INTERFACE I_Pneumatic EXTENDS I_Device

METHOD cancel : BOOL
VAR_INPUT
END_VAR
END_METHOD

METHOD doWait : BOOL
VAR_INPUT
END_VAR
END_METHOD

METHOD doWork : BOOL
VAR_INPUT
END_VAR
END_METHOD

PROPERTY isWait : BOOL
GET
END_GET
END_PROPERTY

PROPERTY isWork : BOOL
GET
END_GET
END_PROPERTY

PROPERTY waitText : STRING(255)
GET
END_GET
SET
END_SET
END_PROPERTY

PROPERTY workText : STRING(255)
GET
END_GET
SET
END_SET
END_PROPERTY

END_INTERFACE

(* stored: Version 1.1.0.1, ProductVersion 3.1.4024.10
   Itf I_Pneumatic: Id {5def5622-ff5f-446d-851f-57a2432c7a0a}
   Method cancel: Id {8ebae174-b4e1-40db-98c4-6a20184f439b}
   Method doWait: Id {807b7b1a-0213-4d92-a090-444ea39660c8}
   Method doWork: Id {b888a43e-f228-4c4e-a392-ad5343d4bdd2}
   Property isWait: Id {d1237558-70e9-44a1-abe1-967740bf8f8e}
   Get Get: Id {ca3f3ba1-7615-4ba6-b68c-5fb93cbb29cb}
   Property isWork: Id {d9ae5c8f-e7ec-4959-bf30-0a123c37b6a8}
   Get Get: Id {cbc7d64f-5cfb-4ac3-a8ee-3dd0d769eaff}
   Property waitText: Id {4c42f9fe-e07d-44e7-af90-b70ff2f04c20}
   Get Get: Id {139db174-8645-4b9a-809b-33fb3059c2cf}
   Set Set: Id {a6a4025c-e12d-476b-a54b-1c7e280e2d5a}
   Property workText: Id {1cfb1efd-4c97-41b3-b6cc-21dffc0ce69a}
   Get Get: Id {29c12924-d4f0-49d8-bd8d-86c3192aed5b}
   Set Set: Id {d99c722d-3e6c-406c-beb8-7971be3dc273} *)
